{attribute 'GeneratedUsingTerminal: APS4322-7000-0017'}
{attribute addProperty BoxType "APS4322-7000-0017"}
{attribute addProperty Id "CommStatusWordAT %I*UINT2DataAT %I*ARRAY[0..3] OF UINT8"}
{attribute addProperty CRC "3146150883"}
{attribute addProperty Size "10"}
TYPE APS_Comm_Inputs_388FE28E EXTENDS InputBase_8311D824 :
STRUCT
	{attribute addProperty Name "CommStatusWord"}
	CommStatusWord AT %I* : UINT;
	{attribute addProperty Name "Data"}
	Data AT %I* : ARRAY[0..3] OF UINT;
END_STRUCT
END_TYPE

(* stored: Version 1.2.0.0, ProductVersion 3.1.4024.11
   DUT APS_Comm_Inputs_388FE28E: Id {1ac85cb5-1e5f-44e2-b662-ed8712ce0832} *)
